FUNCTION_BLOCK FB_Syntax
VAR
    n : INT;
END_VAR

n := n + 1;

METHOD Broken : INT
Broken := n +;
n := 0;
END_METHOD

END_FUNCTION_BLOCK

(* stored: Version 1.1.0.1, ProductVersion 3.1.4024.12
   POU FB_Syntax: Id {5f1c2d9e-0a6b-4c11-9d3e-7a1b2c3d4e80}, SpecialFunc None
   Method Broken: Id {5f1c2d9e-0a6b-4c11-9d3e-7a1b2c3d4e81} *)
